{attribute 'qualified_only'}
{attribute 'strict'}
TYPE ToteStatus:
(
	UNKNOWN 	:= 0,
	EMPTY 		:= 1,
	LOADED		:= 2,
    READY		:= 3
);
END_TYPE

(* stored: Version 1.1.0.1, ProductVersion 3.1.4024.12
   DUT ToteStatus: Id {59d2e8b6-1a92-4a18-8811-9aaf280a7bf4} *)
